# EPICS autosave request: SIS8300App/Db/SIS8300N_settings.req
$(P)$(R)Enable
$(P)$(R)ConvFactor
$(P)$(R)ConvOffset
$(P)$(R)Attenuation
$(P)$(R)DecimFactor
$(P)$(R)DecimOffset
